{attribute 'GeneratedUsingTerminal: EP6002-0002-0016'}
{attribute addProperty BoxType "EP6002-0002-0016"}
{attribute addProperty Id "StatusAT %I*WORD2Data_InAT %I*ARRAY[0..21] OF USINT22"}
{attribute addProperty CRC "3532970676"}
{attribute addProperty Size "24"}
TYPE COM_Inputs_Channel_C252EAC2 :
STRUCT
	{attribute addProperty Name "Status"}
	Status AT %I* : WORD;
	{attribute addProperty Name "Data_In"}
	Data_In AT %I* : ARRAY[0..21] OF USINT;
END_STRUCT
END_TYPE

(* stored: Version 1.2.0.0, ProductVersion 3.1.4024.9
   DUT COM_Inputs_Channel_C252EAC2: Id {c08c84be-2169-4e03-adc3-afcfee705540} *)
